{attribute 'qualified_only'}
VAR_GLOBAL

    BoutonVirtuel : BOOL := FALSE;
	BoutonSelecteur : BOOL := FALSE;
	
	
    LumiereDroite : BOOL := FALSE;
	LumiereGauche : BOOL := FALSE;
	
	CounterLumiereDroiteAllumer : UINT := 0;
	CounterLumiereGaucheAllumer : UINT := 0;
	
	iPushCounter : UINT := 0 ;
	
END_VAR

(* stored: Version 1.1.0.1, ProductVersion 3.1.4024.16
   GVL GVL: Id {53caf463-c901-43aa-a5d3-d1dfaafa4c3e} *)
